TYPE TupleStruct_1:
    STRUCT
        field0: REAL;
        field1: REAL;
    END_STRUCT;
END_TYPE
